PROGRAM MAIN
VAR
	ecat_sim_device_state AT %I* : UINT;
END_VAR

END_PROGRAM

(* stored: Version 1.1.0.1, ProductVersion 3.1.4024.12
   POU MAIN: Id {f8f6236a-c53c-4d5d-bdf4-393a927affae}, SpecialFunc None *)
